// TIA Portal V18 export
VAR_GLOBAL   // PLC tag table "Ready"
   Ready_TF_Pump_Aeration_Clarifier_01 AT %I7.4 : Bool;
   Ready_TF_Pump_Aeration_Clarifier_02 AT %I7.5 : Bool;
   Ready_Suction_Pump_01 AT %I4.5 : Bool;
   Ready_Suction_Pump_02 AT %I4.6 : Bool;
   Ready_Suction_Pump_03 AT %I4.7 : Bool;
   Ready_Suction_Pump_04 AT %I5.0 : Bool;
   Ready_Suction_Pump_05 AT %I5.1 : Bool;
   Ready_Suction_Pump_06 AT %I5.2 : Bool;
   Ready_Suction_Pump_07 AT %I5.3 : Bool;
   Ready_Suction_Pump_08 AT %I5.4 : Bool;
   Ready_Backwash_Pump_01 AT %I5.5 : Bool;
   Ready_Backwash_Pump_02 AT %I5.6 : Bool;
   Ready_Backwash_Pump_03 AT %I5.7 : Bool;
   Ready_Backwash_Pump_04 AT %I6.0 : Bool;
   Ready_Backwash_Pump_05 AT %I6.1 : Bool;
   Ready_MBR_Aeration_01 AT %I6.2 : Bool;
   Ready_MBR_Aeration_02 AT %I6.3 : Bool;
   Ready_Chlorine_Dosing_Pump AT %I6.4 : Bool;
   Ready_Chlorine_Chemical_Agitator AT %I6.5 : Bool;
   Ready_Solid_TF_Clarifier AT %I6.6 : Bool;
   Ready_UV_1P_01 AT %I6.7 : Bool;
   Ready_UV_1P_02 AT %I7.0 : Bool;
   Ready_UV_1P_03 AT %I7.1 : Bool;
   Ready_TF_Pump_CSAS_B_01 AT %I7.2 : Bool;
   Ready_TF_Pump_CSAS_B_02 AT %I7.3 : Bool;
   Ready_TF_Pump_RWT_MMF_01 AT %I7.6 : Bool;
   Ready_TF_Pump_RWT_MMF_02 AT %I7.7 : Bool;
   Ready_PAC_Floculant_Dosing_Pump AT %I8.0 : Bool;
   Ready_TF_Pump_Waterpool_Buffer_01_Main AT %I8.1 : Bool;
   Ready_TF_Pump_Waterpool_Buffer_01_Delta AT %I8.2 : Bool;
   Ready_TF_Pump_Waterpool_Buffer_01_Star AT %I8.3 : Bool;
   Ready_TF_Pump_Waterpool_Buffer_02_Main AT %I8.4 : Bool;
   Ready_TF_Pump_Waterpool_Buffer_02_Delta AT %I8.5 : Bool;
   Ready_TF_Pump_Waterpool_Buffer_02_Star AT %I8.6 : Bool;
END_VAR
